FUNCTION_BLOCK FB_MqttSubClient
VAR_INPUT
	stMqttConnect : ST_MqttConnect;
	TopicToSubscribe : STRING(255);
	fbMqttMessageQueue: FB_IotMqttMessageQueue;
	fbMqttMessage: FB_IotMqttMessage;
END_VAR
VAR_OUTPUT
	bGetValue : BOOL;
END_VAR
VAR
	fbMqttClient: FB_IotMqttClient;
	Subscribed:BOOL;
    ReceivingTopic:STRING(255);
	ReceivingData:STRING(255);
END_VAR

fbMqttClient.sClientId := stMqttConnect.sClientID;
fbMqttClient.sHostName := stMqttConnect.sHostName;
fbMqttClient.nHostPort := stMqttConnect.nHostPort;
fbMqttClient.sTopicPrefix := stMqttConnect.sTopicPrefix;
fbMqttClient.nKeepAlive := stMqttConnect.nKeepAlive;
fbMqttClient.ipMessageQueue := fbMqttMessageQueue;

fbMqttClient.Execute(bConnect :=TRUE);
 
IF fbMqttClient.bConnected THEN
    IF NOT Subscribed THEN
        Subscribed := fbMqttClient.Subscribe(sTopic:=TopicToSubscribe,
        eQoS:=TcIotMqttQos.AtMostOnceDelivery);
    END_IF
END_IF
 

IF fbMqttMessageQueue.Dequeue(fbMessage:=fbMqttMessage) THEN
	 fbMqttMessage.GetTopic(pTopic:=ADR(ReceivingTopic), nTopicSize:=SIZEOF(ReceivingTopic) );
	 fbMqttMessage.GetPayload(pPayload:=ADR(ReceivingData), nPayloadSize:=SIZEOF(ReceivingData), bSetNullTermination:=FALSE);
END_IF


IF ReceivingData = 'truee' THEN
	bGetValue := TRUE;
ELSE
	bGetValue := FALSE;
END_IF

END_FUNCTION_BLOCK

(* stored: Version 1.1.0.1, ProductVersion 3.1.4024.15
   POU FB_MqttSubClient: Id {b22460df-a923-4c27-ad81-ff8dd7a49e1a}, SpecialFunc None *)
